// TIA Portal V16 export
// export: Created 2021-04-06T19:52:19.2596619Z, ExportSetting WithDefaults, DisplayName Totally Integrated Automation Portal, DisplayVersion V16, DisplayName TIA Portal Version Control Interface, DisplayVersion V16, DisplayName TIA Portal Openness, DisplayVersion V16, DisplayName STEP 7 Professional, DisplayVersion V16, DisplayName STEP 7 Safety, DisplayVersion V16, DisplayName WinCC Unified SCADA Engineering System, DisplayVersion V16
TYPE "outConv"
// stored: IsFailsafeCompliant false
   STRUCT
      isUpInBegin : Bool;   // направление вращения для упаковки
      isUseInBegin : Bool;   // использовать ли конвейер для упаковки
      isUpInEnd : Bool;   // направления вращения при очистке
      setWeightPack : Real;   // вес упаковки
      currentWeightPack : Real;   // текущий вес упаковки
      currentErrorMeasure : Real;   // текущая погрешность
      isWorkConv : Bool;   // работа конвейера
      isAlarmConv : Bool;   // авария конвейера
      isReadyPackingMachine : Bool;   // сигнал готовности упаковочной машины
      isReadyDozaPackingMachine : Bool;   // сигнал доза упаковочной машины
      manStartOutConv : Bool;   // ручн - запуск конвейера
      stateConvInt : Int;   // состояние конвейера
      manIsUpConv : Bool;   // ручн - конв вперед\назад
   END_STRUCT;
END_TYPE
